(* PLC project Cell Example , CTH FIX1 1.0, author CTH SS2 *)
(* stored: creationDateTime 2009-04-27T15:46:22, companyURL www.chalmers.se, language en-US, organization SS2, modificationDateTime 2008-04-09T20:25:24, version 1.0 *)

PROGRAM EOP10_a
  VAR_EXTERNAL
    Op_10_start : BOOL := false;
    C1C2C1_in_position_empty : BOOL := false;
    C1C2C2_in_off : BOOL := false;
    Op_10_end : BOOL := false;
  END_VAR
  VAR  (* added by the conversion: wires and edge detectors of the diagram *)
    _AND4_OUT : BOOL;
    _AND9_OUT : BOOL;
  END_VAR

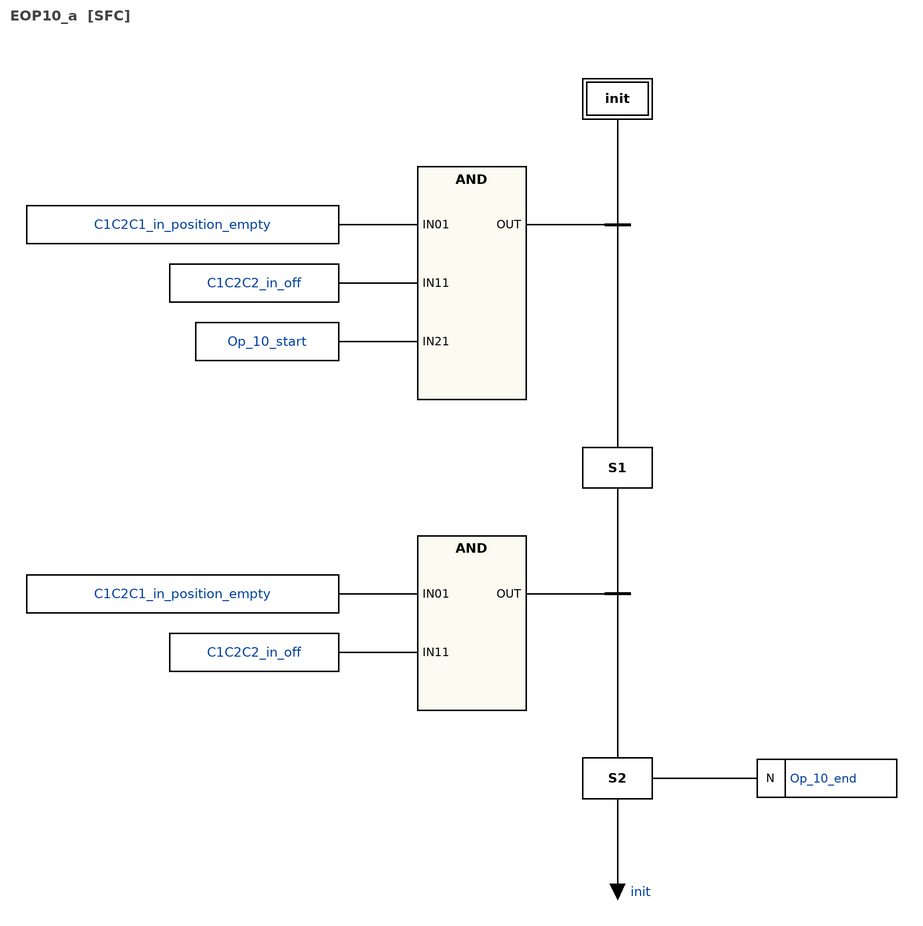
INITIAL_STEP init:
  COMPUTE_FUNCTION_BLOCKS(S);
END_STEP
TRANSITION FROM init TO S1
  := _AND4_OUT;
END_TRANSITION
STEP S1:
END_STEP
TRANSITION FROM S1 TO S2
  := _AND9_OUT;
END_TRANSITION
STEP S2:
  Op_10_end(N);
END_STEP
ACTION COMPUTE_FUNCTION_BLOCKS:  (* blocks drawn on the SFC sheet *)
  _AND4_OUT := C1C2C1_in_position_empty AND C1C2C2_in_off AND Op_10_start;
  _AND9_OUT := C1C2C1_in_position_empty AND C1C2C2_in_off;
END_ACTION
END_PROGRAM

PROGRAM EOP10_b
  VAR_EXTERNAL
    Op_10_start : BOOL := false;
    C1C2C1_in_part_in_position : BOOL := false;
    C1C2C2_in_on : BOOL := false;
    Op_10_end : BOOL := false;
  END_VAR
  VAR  (* added by the conversion: wires and edge detectors of the diagram *)
    _AND4_OUT : BOOL;
    _AND9_OUT : BOOL;
  END_VAR

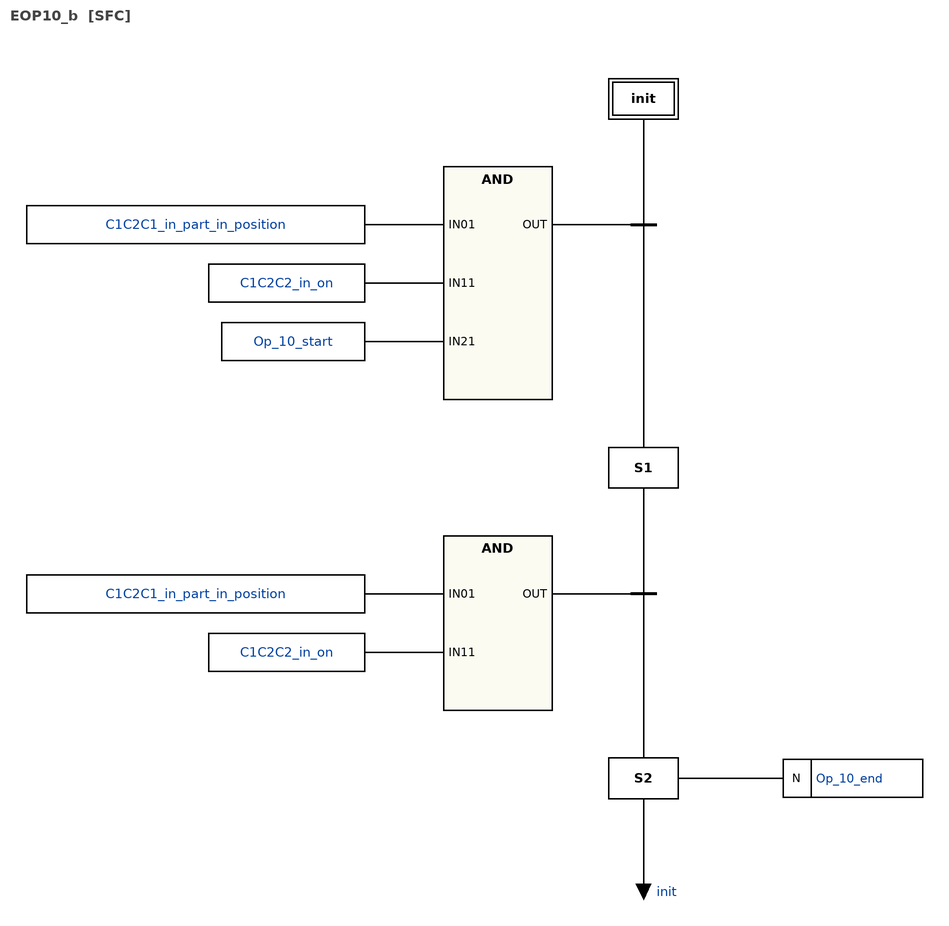
INITIAL_STEP init:
  COMPUTE_FUNCTION_BLOCKS(S);
END_STEP
TRANSITION FROM init TO S1
  := _AND4_OUT;
END_TRANSITION
STEP S1:
END_STEP
TRANSITION FROM S1 TO S2
  := _AND9_OUT;
END_TRANSITION
STEP S2:
  Op_10_end(N);
END_STEP
ACTION COMPUTE_FUNCTION_BLOCKS:  (* blocks drawn on the SFC sheet *)
  _AND4_OUT := C1C2C1_in_part_in_position AND C1C2C2_in_on AND Op_10_start;
  _AND9_OUT := C1C2C1_in_part_in_position AND C1C2C2_in_on;
END_ACTION
END_PROGRAM

PROGRAM EOP11
  VAR_EXTERNAL
    Op_11_start : BOOL := false;
    TRUE_VAR : BOOL := true;
    C1C2_book_zone_1 : BOOL := false;
    C1C2_zone_1_booked : BOOL := false;
    C1C2C1_goto_part_in_position : BOOL := false;
    C1C2C2_goto_on : BOOL := false;
    C1C2C1_in_part_in_position : BOOL := false;
    C1C2C2_in_on : BOOL := false;
    C1C2_unbook_zone_1 : BOOL := false;
    Op_11_end : BOOL := false;
  END_VAR
  VAR  (* added by the conversion: wires and edge detectors of the diagram *)
    _AND14_OUT : BOOL;
    _AND21_OUT : BOOL;
  END_VAR

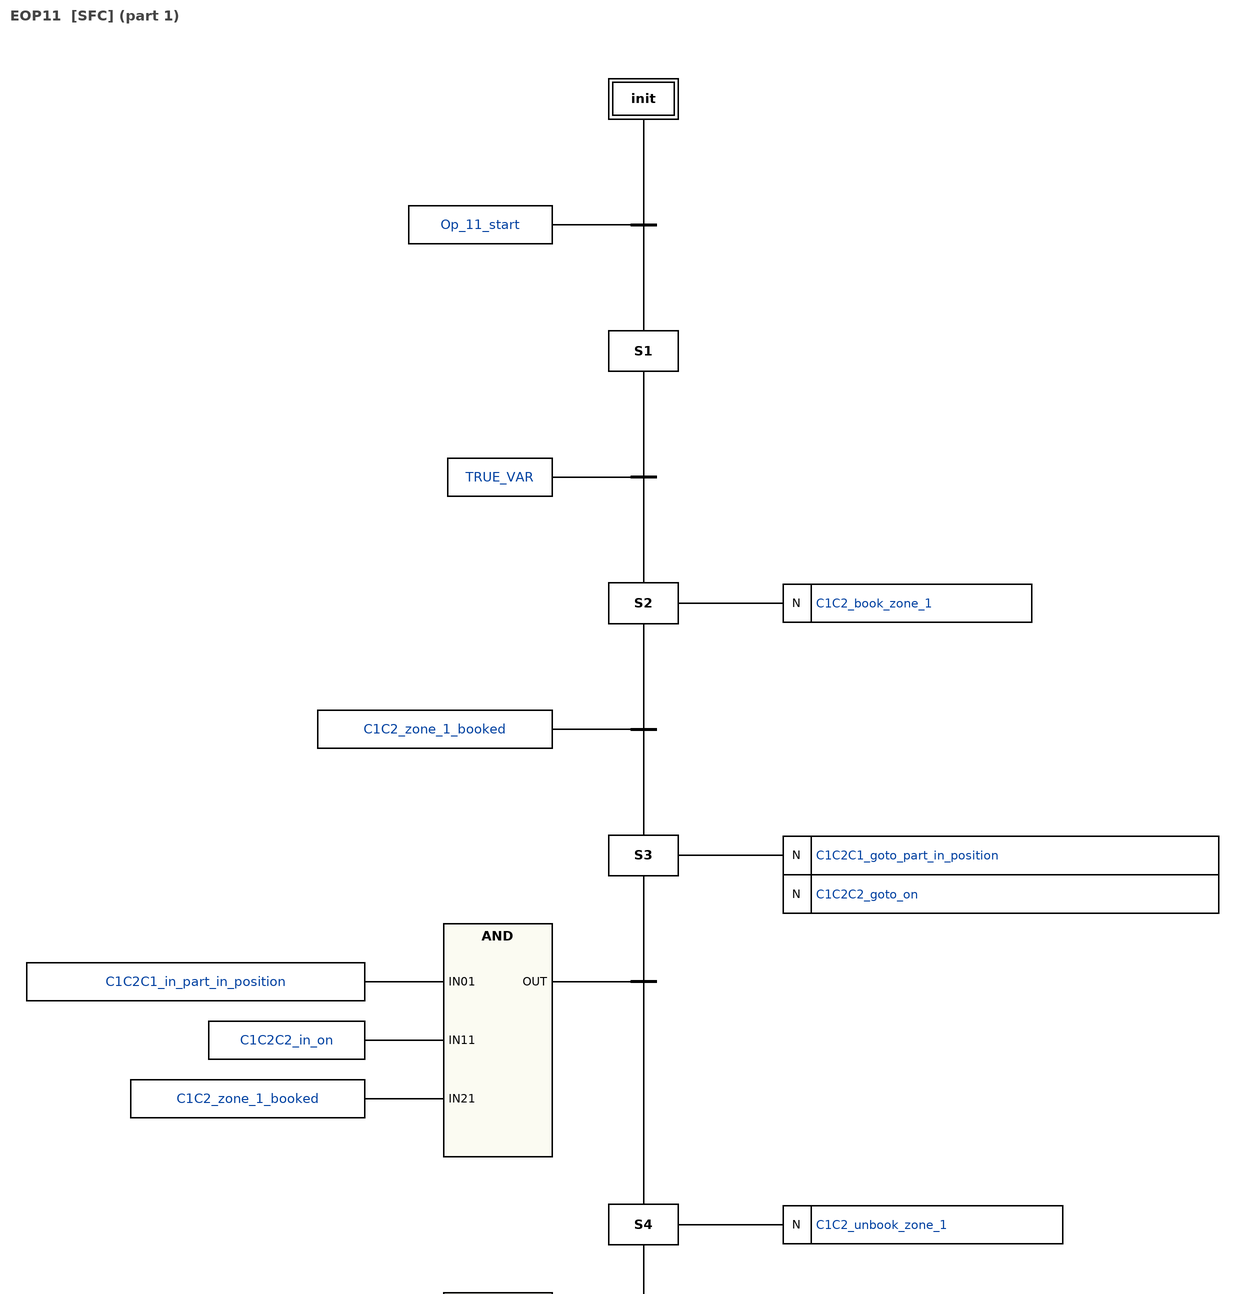
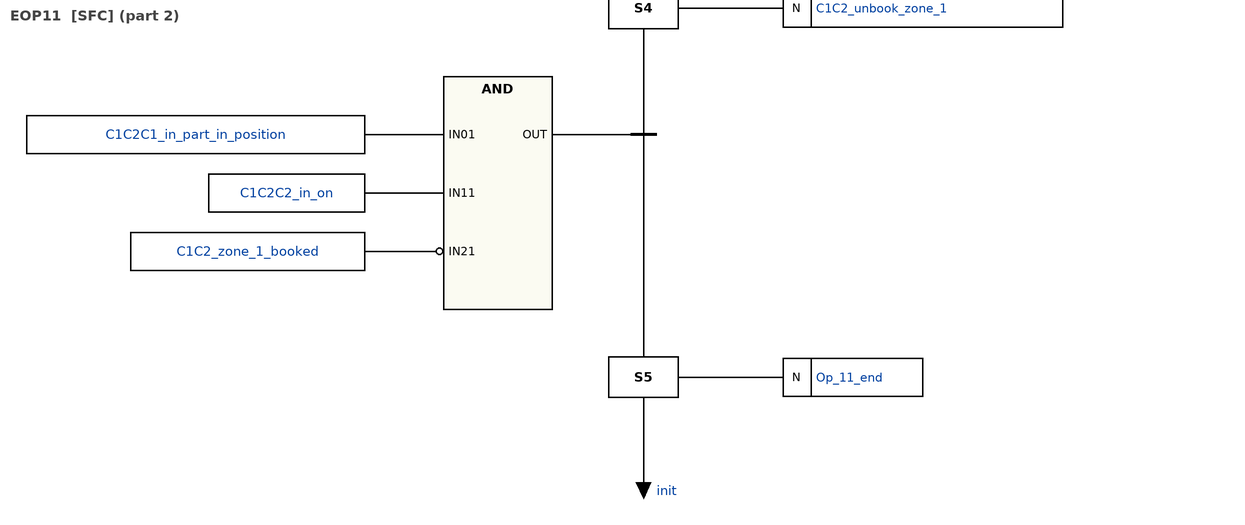
INITIAL_STEP init:
  COMPUTE_FUNCTION_BLOCKS(S);
END_STEP
TRANSITION FROM init TO S1
  := Op_11_start;
END_TRANSITION
STEP S1:
END_STEP
TRANSITION FROM S1 TO S2
  := TRUE_VAR;
END_TRANSITION
STEP S2:
  C1C2_book_zone_1(N);
END_STEP
TRANSITION FROM S2 TO S3
  := C1C2_zone_1_booked;
END_TRANSITION
STEP S3:
  C1C2C1_goto_part_in_position(N);
  C1C2C2_goto_on(N);
END_STEP
TRANSITION FROM S3 TO S4
  := _AND14_OUT;
END_TRANSITION
STEP S4:
  C1C2_unbook_zone_1(N);
END_STEP
TRANSITION FROM S4 TO S5
  := _AND21_OUT;
END_TRANSITION
STEP S5:
  Op_11_end(N);
END_STEP
ACTION COMPUTE_FUNCTION_BLOCKS:  (* blocks drawn on the SFC sheet *)
  _AND14_OUT := C1C2C1_in_part_in_position AND C1C2C2_in_on AND C1C2_zone_1_booked;
  _AND21_OUT := C1C2C1_in_part_in_position AND C1C2C2_in_on AND NOT C1C2_zone_1_booked;
END_ACTION
END_PROGRAM

PROGRAM EOP12
  VAR_EXTERNAL
    Op_12_start : BOOL := false;
    TRUE_VAR : BOOL := true;
    C1C2C1_goto_position_empty : BOOL := false;
    C1C2C2_goto_off : BOOL := false;
    C1C2C1_in_position_empty : BOOL := false;
    C1C2C2_in_off : BOOL := false;
    Op_12_end : BOOL := false;
  END_VAR
  VAR  (* added by the conversion: wires and edge detectors of the diagram *)
    _AND10_OUT : BOOL;
  END_VAR

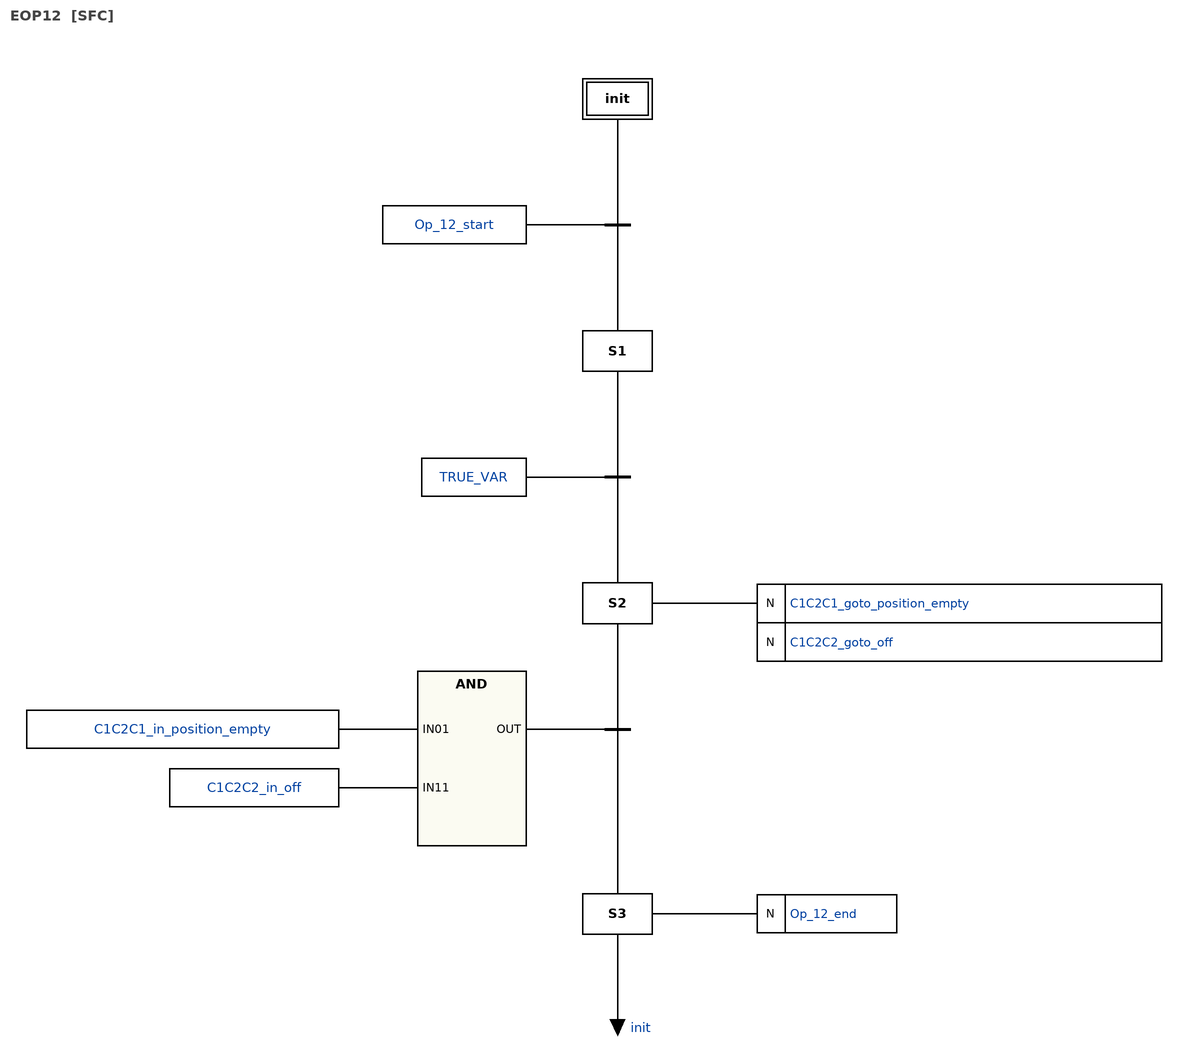
INITIAL_STEP init:
  COMPUTE_FUNCTION_BLOCKS(S);
END_STEP
TRANSITION FROM init TO S1
  := Op_12_start;
END_TRANSITION
STEP S1:
END_STEP
TRANSITION FROM S1 TO S2
  := TRUE_VAR;
END_TRANSITION
STEP S2:
  C1C2C1_goto_position_empty(N);
  C1C2C2_goto_off(N);
END_STEP
TRANSITION FROM S2 TO S3
  := _AND10_OUT;
END_TRANSITION
STEP S3:
  Op_12_end(N);
END_STEP
ACTION COMPUTE_FUNCTION_BLOCKS:  (* blocks drawn on the SFC sheet *)
  _AND10_OUT := C1C2C1_in_position_empty AND C1C2C2_in_off;
END_ACTION
END_PROGRAM

PROGRAM EOP20
  VAR_EXTERNAL
    C1R1_Op20_exe_start : BOOL := false;
    C1R1_in_inital : BOOL := false;
    C1R1_Op20_exe : BOOL := false;
    C1R1_Op20_done : BOOL := false;
  END_VAR

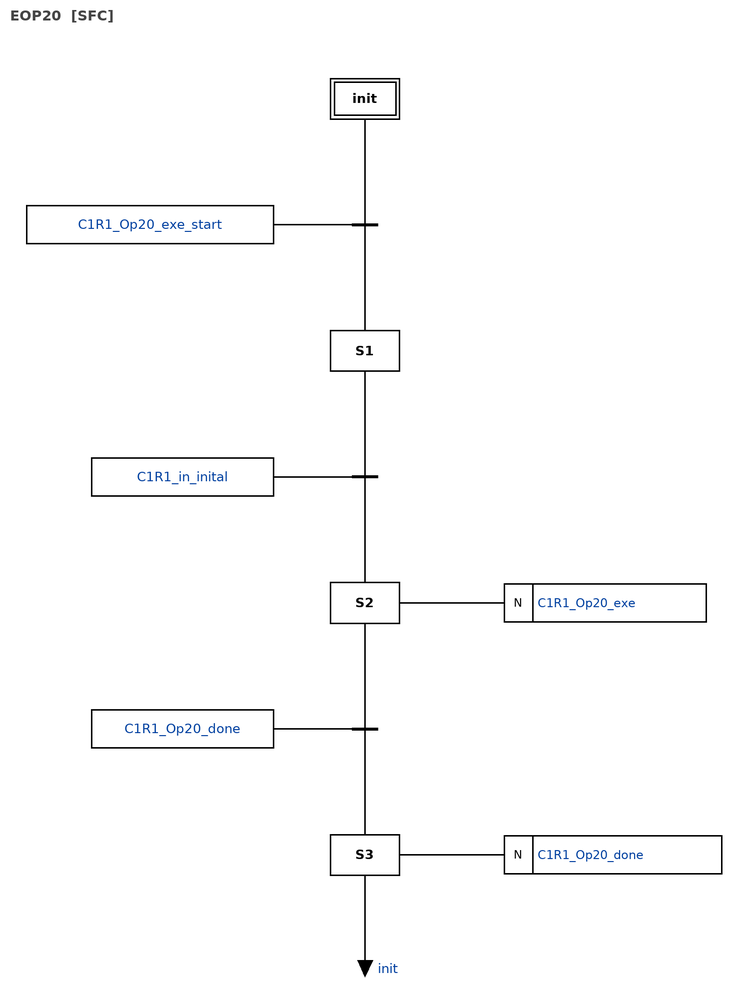
INITIAL_STEP init:
END_STEP
TRANSITION FROM init TO S1
  := C1R1_Op20_exe_start;
END_TRANSITION
STEP S1:
END_STEP
TRANSITION FROM S1 TO S2
  := C1R1_in_inital;
END_TRANSITION
STEP S2:
  C1R1_Op20_exe(N);
END_STEP
TRANSITION FROM S2 TO S3
  := C1R1_Op20_done;
END_TRANSITION
STEP S3:
  C1R1_Op20_done(N);
END_STEP
END_PROGRAM

PROGRAM EOP21
  VAR_EXTERNAL
    C1R1_Op21_exe_start : BOOL := false;
    TRUE_VAR : BOOL := true;
    C1R1_book_zone_1 : BOOL := false;
    C1R1_zone_1_booked : BOOL := false;
    C1R1_Op21_exe : BOOL := false;
    C1R1_Op21_done : BOOL := false;
    C1R1_unbook_zone_1 : BOOL := false;
  END_VAR
  VAR  (* added by the conversion: wires and edge detectors of the diagram *)
    _NOT19_OUT : BOOL;
  END_VAR

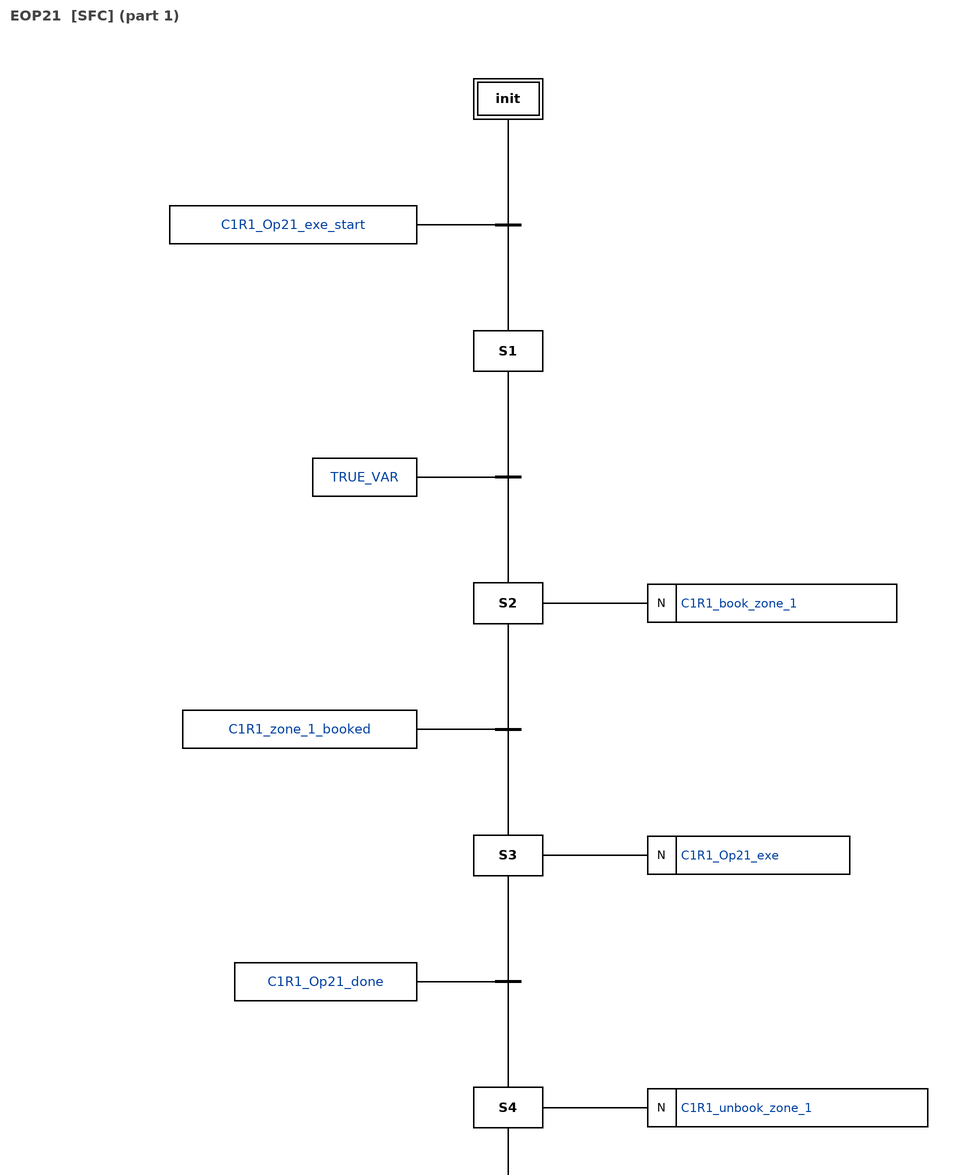
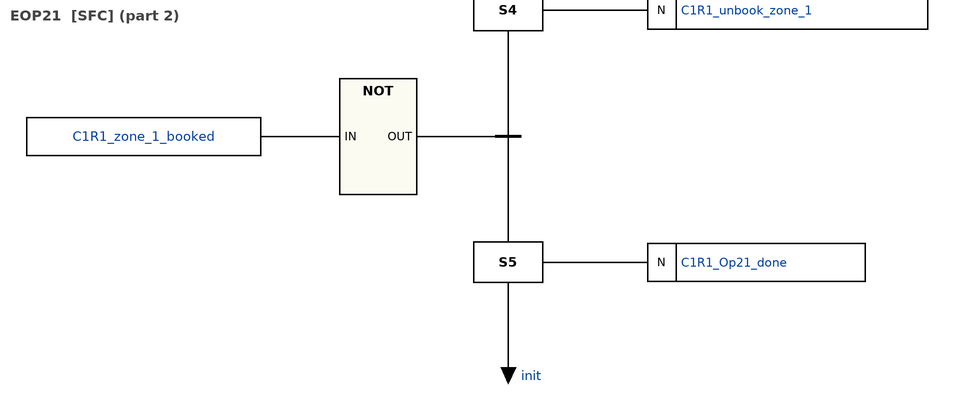
INITIAL_STEP init:
  COMPUTE_FUNCTION_BLOCKS(S);
END_STEP
TRANSITION FROM init TO S1
  := C1R1_Op21_exe_start;
END_TRANSITION
STEP S1:
END_STEP
TRANSITION FROM S1 TO S2
  := TRUE_VAR;
END_TRANSITION
STEP S2:
  C1R1_book_zone_1(N);
END_STEP
TRANSITION FROM S2 TO S3
  := C1R1_zone_1_booked;
END_TRANSITION
STEP S3:
  C1R1_Op21_exe(N);
END_STEP
TRANSITION FROM S3 TO S4
  := C1R1_Op21_done;
END_TRANSITION
STEP S4:
  C1R1_unbook_zone_1(N);
END_STEP
TRANSITION FROM S4 TO S5
  := _NOT19_OUT;
END_TRANSITION
STEP S5:
  C1R1_Op21_done(N);
END_STEP
ACTION COMPUTE_FUNCTION_BLOCKS:  (* blocks drawn on the SFC sheet *)
  _NOT19_OUT := NOT C1R1_zone_1_booked;
END_ACTION
END_PROGRAM

PROGRAM EOP22
  VAR_EXTERNAL
    C1R1_Op22_exe_start : BOOL := false;
    TRUE_VAR : BOOL := true;
    C1R1_book_zone_1 : BOOL := false;
    C1R1_zone_1_booked : BOOL := false;
    C1R1_Op22_exe : BOOL := false;
    C1R1_Op22_done : BOOL := false;
  END_VAR

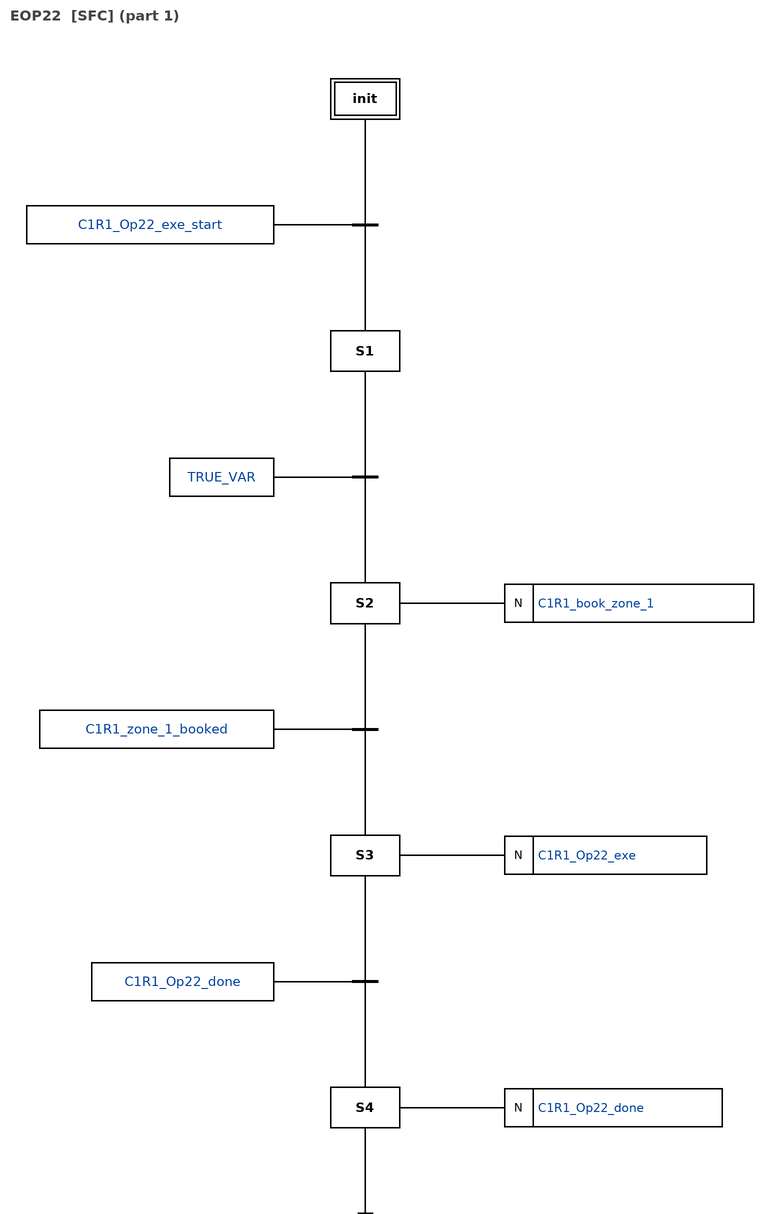
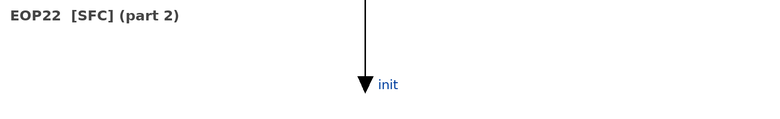
INITIAL_STEP init:
END_STEP
TRANSITION FROM init TO S1
  := C1R1_Op22_exe_start;
END_TRANSITION
STEP S1:
END_STEP
TRANSITION FROM S1 TO S2
  := TRUE_VAR;
END_TRANSITION
STEP S2:
  C1R1_book_zone_1(N);
END_STEP
TRANSITION FROM S2 TO S3
  := C1R1_zone_1_booked;
END_TRANSITION
STEP S3:
  C1R1_Op22_exe(N);
END_STEP
TRANSITION FROM S3 TO S4
  := C1R1_Op22_done;
END_TRANSITION
STEP S4:
  C1R1_Op22_done(N);
END_STEP
END_PROGRAM

PROGRAM EOP23
  VAR_EXTERNAL
    C1R1_Op23_exe_start : BOOL := false;
    TRUE_VAR : BOOL := true;
    C1R1_book_zone_2 : BOOL := false;
    C1R1_zone_2_booked : BOOL := false;
    C1R1_Op23_exe : BOOL := false;
    C1R1_Op23_done : BOOL := false;
    C1R1_unbook_zone_2 : BOOL := false;
  END_VAR
  VAR  (* added by the conversion: wires and edge detectors of the diagram *)
    _NOT19_OUT : BOOL;
  END_VAR

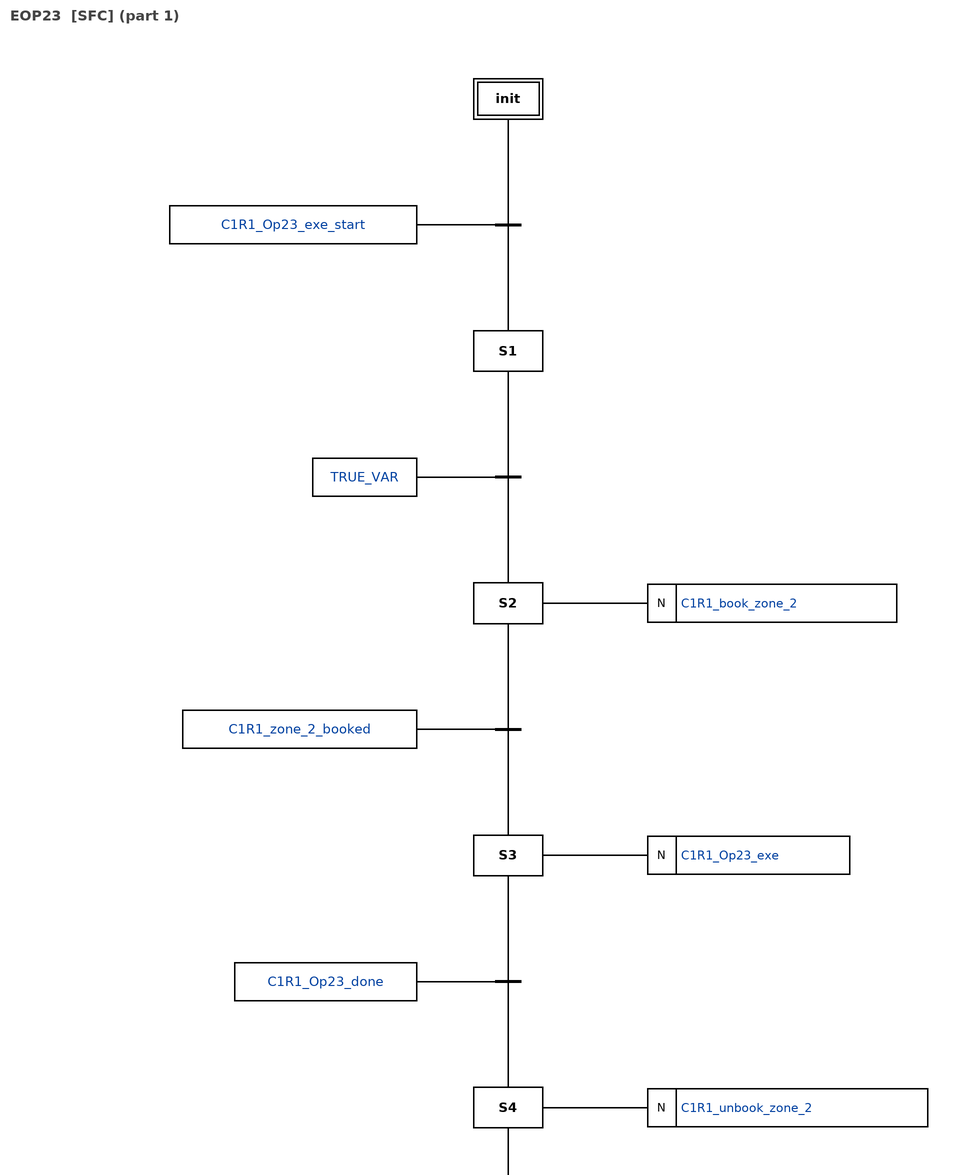
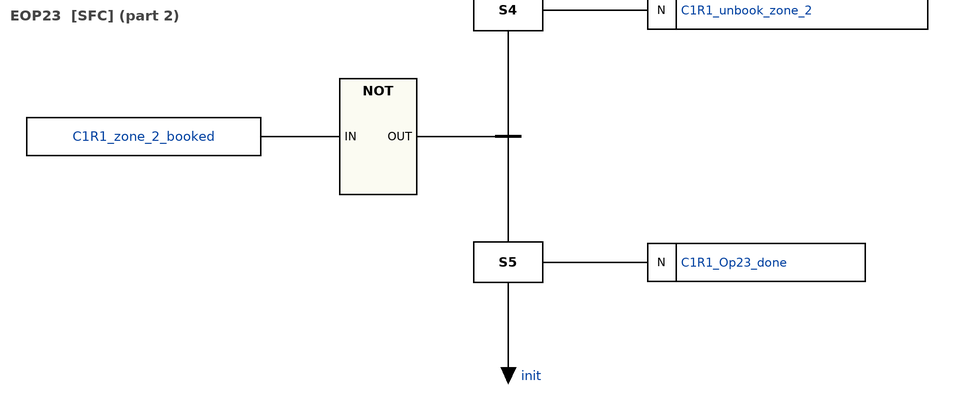
INITIAL_STEP init:
  COMPUTE_FUNCTION_BLOCKS(S);
END_STEP
TRANSITION FROM init TO S1
  := C1R1_Op23_exe_start;
END_TRANSITION
STEP S1:
END_STEP
TRANSITION FROM S1 TO S2
  := TRUE_VAR;
END_TRANSITION
STEP S2:
  C1R1_book_zone_2(N);
END_STEP
TRANSITION FROM S2 TO S3
  := C1R1_zone_2_booked;
END_TRANSITION
STEP S3:
  C1R1_Op23_exe(N);
END_STEP
TRANSITION FROM S3 TO S4
  := C1R1_Op23_done;
END_TRANSITION
STEP S4:
  C1R1_unbook_zone_2(N);
END_STEP
TRANSITION FROM S4 TO S5
  := _NOT19_OUT;
END_TRANSITION
STEP S5:
  C1R1_Op23_done(N);
END_STEP
ACTION COMPUTE_FUNCTION_BLOCKS:  (* blocks drawn on the SFC sheet *)
  _NOT19_OUT := NOT C1R1_zone_2_booked;
END_ACTION
END_PROGRAM

PROGRAM EOP24
  VAR_EXTERNAL
    C1R1_Op24_exe_start : BOOL := false;
    TRUE_VAR : BOOL := true;
    C1R1_book_zone_3 : BOOL := false;
    C1R1_zone_3_booked : BOOL := false;
    C1R1_Op24_exe : BOOL := false;
    C1R1_Op24_done : BOOL := false;
    C1R1_unbook_zone_3 : BOOL := false;
  END_VAR
  VAR  (* added by the conversion: wires and edge detectors of the diagram *)
    _NOT19_OUT : BOOL;
  END_VAR

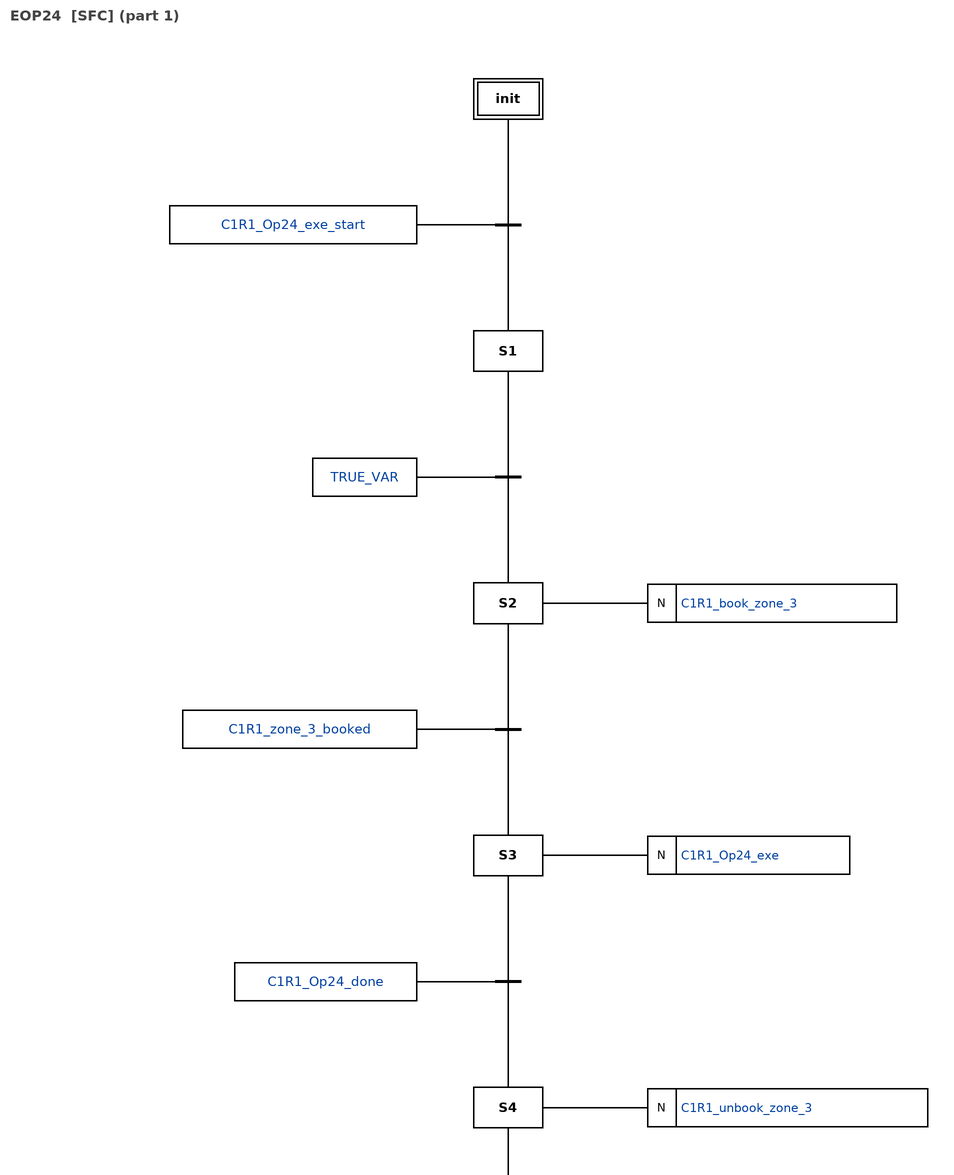
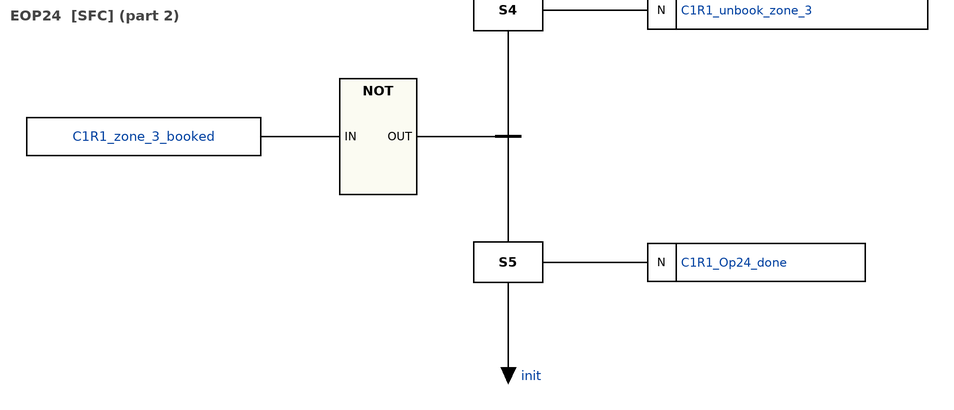
INITIAL_STEP init:
  COMPUTE_FUNCTION_BLOCKS(S);
END_STEP
TRANSITION FROM init TO S1
  := C1R1_Op24_exe_start;
END_TRANSITION
STEP S1:
END_STEP
TRANSITION FROM S1 TO S2
  := TRUE_VAR;
END_TRANSITION
STEP S2:
  C1R1_book_zone_3(N);
END_STEP
TRANSITION FROM S2 TO S3
  := C1R1_zone_3_booked;
END_TRANSITION
STEP S3:
  C1R1_Op24_exe(N);
END_STEP
TRANSITION FROM S3 TO S4
  := C1R1_Op24_done;
END_TRANSITION
STEP S4:
  C1R1_unbook_zone_3(N);
END_STEP
TRANSITION FROM S4 TO S5
  := _NOT19_OUT;
END_TRANSITION
STEP S5:
  C1R1_Op24_done(N);
END_STEP
ACTION COMPUTE_FUNCTION_BLOCKS:  (* blocks drawn on the SFC sheet *)
  _NOT19_OUT := NOT C1R1_zone_3_booked;
END_ACTION
END_PROGRAM

PROGRAM EOP30
  VAR_EXTERNAL
    Op_30_start : BOOL := false;
    C1F1C1_in_home : BOOL := false;
    C1F1C2_in_locked : BOOL := false;
    C1F1C3_in_open : BOOL := false;
    C1F1C4_in_off : BOOL := false;
    Op_30_end : BOOL := false;
  END_VAR
  VAR  (* added by the conversion: wires and edge detectors of the diagram *)
    _AND6_OUT : BOOL;
  END_VAR

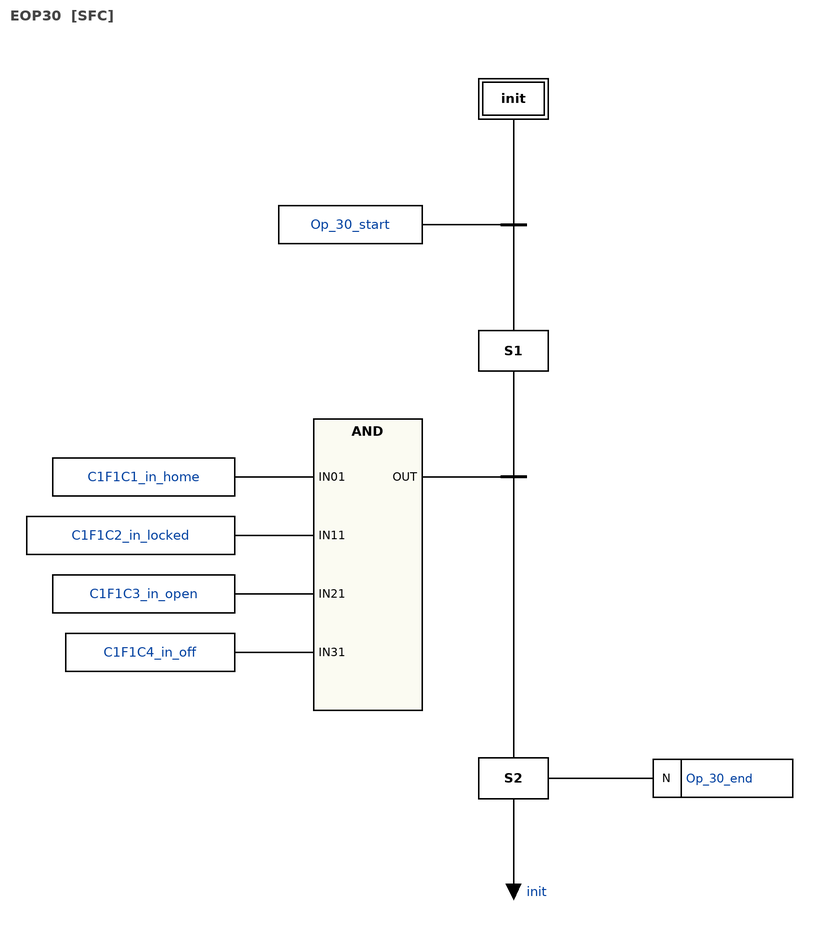
INITIAL_STEP init:
  COMPUTE_FUNCTION_BLOCKS(S);
END_STEP
TRANSITION FROM init TO S1
  := Op_30_start;
END_TRANSITION
STEP S1:
END_STEP
TRANSITION FROM S1 TO S2
  := _AND6_OUT;
END_TRANSITION
STEP S2:
  Op_30_end(N);
END_STEP
ACTION COMPUTE_FUNCTION_BLOCKS:  (* blocks drawn on the SFC sheet *)
  _AND6_OUT := C1F1C1_in_home AND C1F1C2_in_locked AND C1F1C3_in_open AND C1F1C4_in_off;
END_ACTION
END_PROGRAM

PROGRAM EOP31
  VAR_EXTERNAL
    Op_31_start : BOOL := false;
    TRUE_VAR : BOOL := true;
    Op_31_end : BOOL := false;
  END_VAR

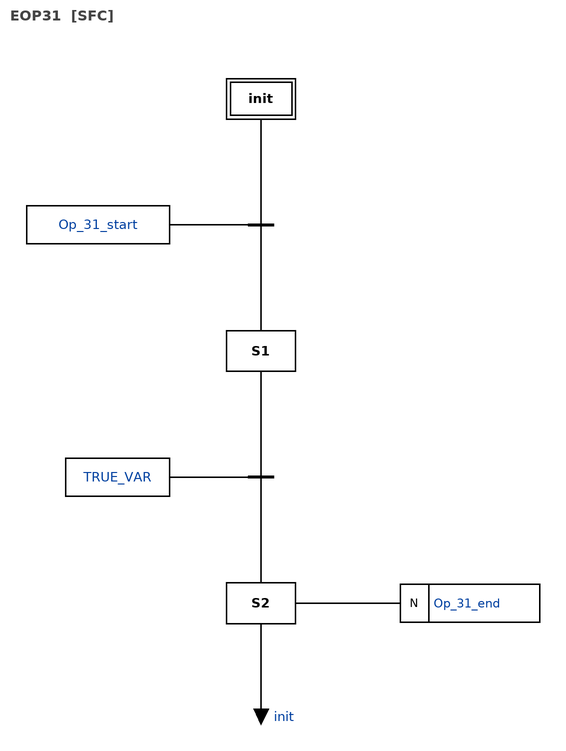
INITIAL_STEP init:
END_STEP
TRANSITION FROM init TO S1
  := Op_31_start;
END_TRANSITION
STEP S1:
END_STEP
TRANSITION FROM S1 TO S2
  := TRUE_VAR;
END_TRANSITION
STEP S2:
  Op_31_end(N);
END_STEP
END_PROGRAM

PROGRAM EOP32
  VAR_EXTERNAL
    Op_32_start : BOOL := false;
    TRUE_VAR : BOOL := true;
    C1F1C1_goto_home : BOOL := false;
    C1F1C2_goto_locked : BOOL := false;
    C1F1C3_goto_close : BOOL := false;
    C1F1C4_goto_on : BOOL := false;
    C1F1C1_in_home : BOOL := false;
    C1F1C2_in_locked : BOOL := false;
    C1F1C3_in_close : BOOL := false;
    C1F1C4_in_on : BOOL := false;
    Op_32_end : BOOL := false;
  END_VAR
  VAR  (* added by the conversion: wires and edge detectors of the diagram *)
    _AND10_OUT : BOOL;
  END_VAR

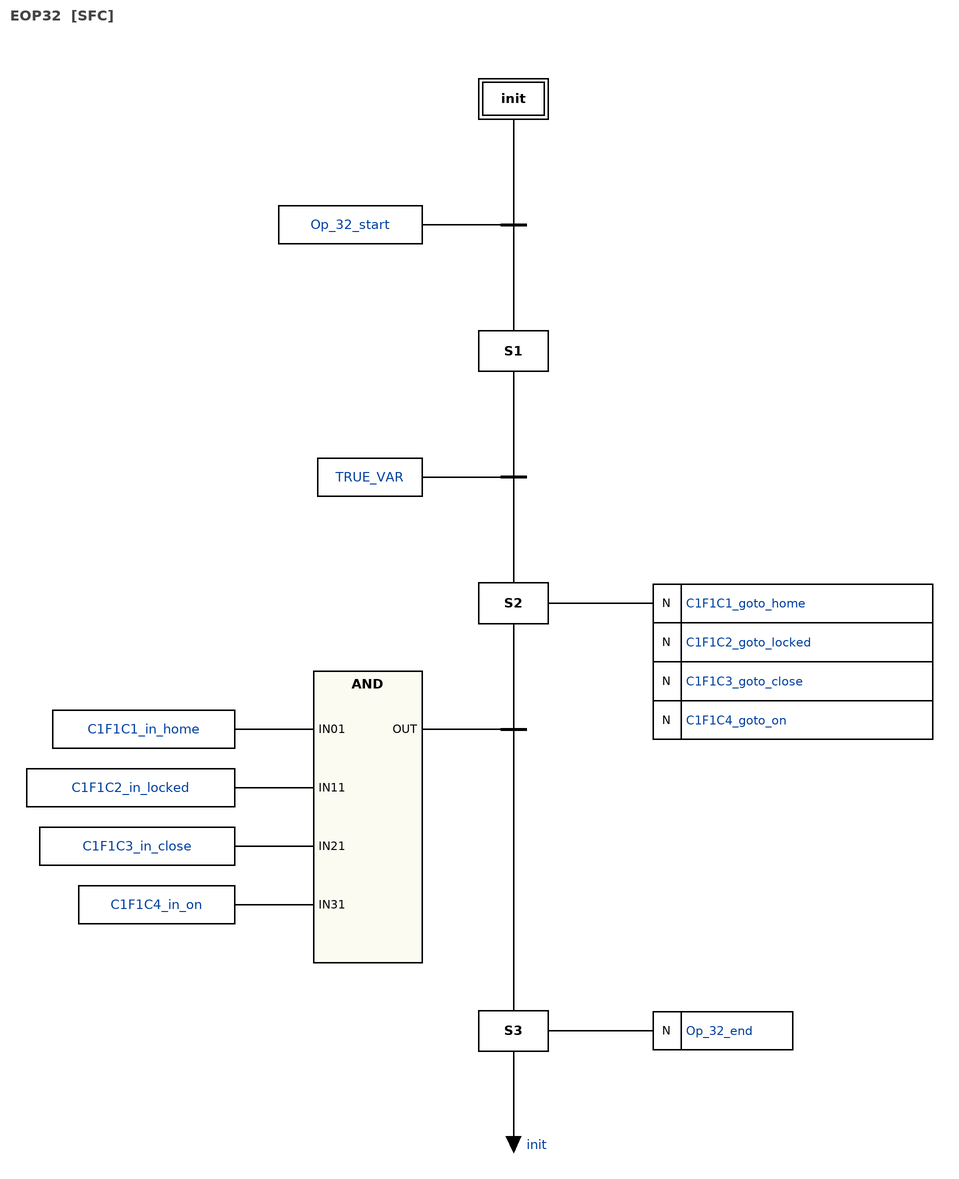
INITIAL_STEP init:
  COMPUTE_FUNCTION_BLOCKS(S);
END_STEP
TRANSITION FROM init TO S1
  := Op_32_start;
END_TRANSITION
STEP S1:
END_STEP
TRANSITION FROM S1 TO S2
  := TRUE_VAR;
END_TRANSITION
STEP S2:
  C1F1C1_goto_home(N);
  C1F1C2_goto_locked(N);
  C1F1C3_goto_close(N);
  C1F1C4_goto_on(N);
END_STEP
TRANSITION FROM S2 TO S3
  := _AND10_OUT;
END_TRANSITION
STEP S3:
  Op_32_end(N);
END_STEP
ACTION COMPUTE_FUNCTION_BLOCKS:  (* blocks drawn on the SFC sheet *)
  _AND10_OUT := C1F1C1_in_home AND C1F1C2_in_locked AND C1F1C3_in_close AND C1F1C4_in_on;
END_ACTION
END_PROGRAM

PROGRAM EOP33
  VAR_EXTERNAL
    Op_33_start : BOOL := false;
    TRUE_VAR : BOOL := true;
    C1F1C1_goto_home : BOOL := false;
    C1F1C2_goto_unlocked : BOOL := false;
    C1F1C3_goto_close : BOOL := false;
    C1F1C4_goto_on : BOOL := false;
    C1F1_book_zone_2 : BOOL := false;
    C1F1_book_zone_3 : BOOL := false;
    C1F1C1_in_home : BOOL := false;
    C1F1C2_in_unlocked : BOOL := false;
    C1F1C3_in_close : BOOL := false;
    C1F1C4_in_on : BOOL := false;
    C1F1_zone_2_booked : BOOL := false;
    C1F1_zone_3_booked : BOOL := false;
    C1F1C1_goto_work_pos : BOOL := false;
    C1F1C1_in_work_pos : BOOL := false;
    C1F1C2_goto_locked : BOOL := false;
    C1F1_unbook_zone_3 : BOOL := false;
    C1F1C2_in_locked : BOOL := false;
    Op_33_end : BOOL := false;
  END_VAR
  VAR  (* added by the conversion: wires and edge detectors of the diagram *)
    _AND10_OUT : BOOL;
    _AND20_OUT : BOOL;
    _AND30_OUT : BOOL;
  END_VAR

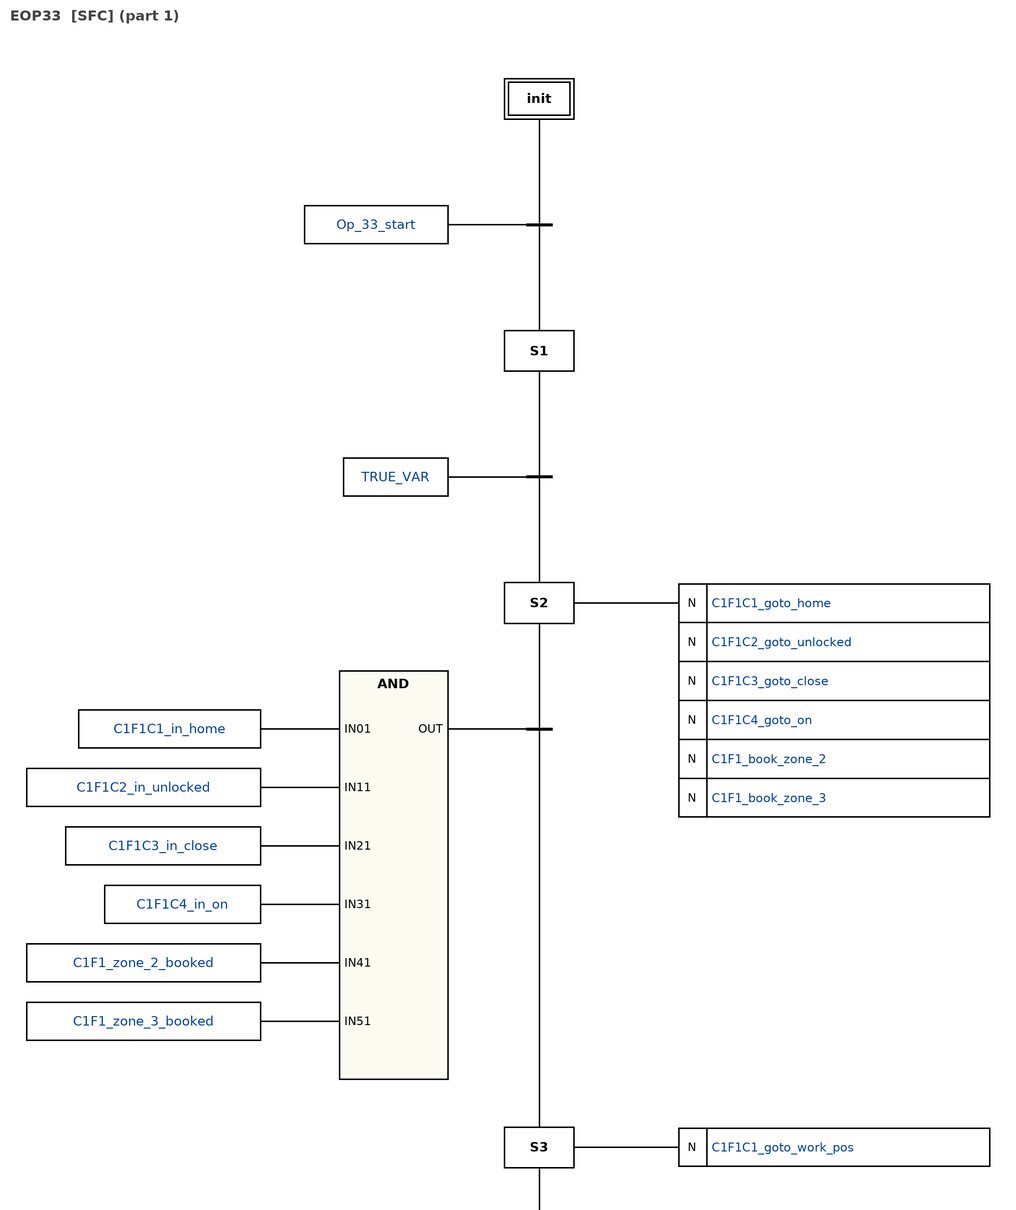
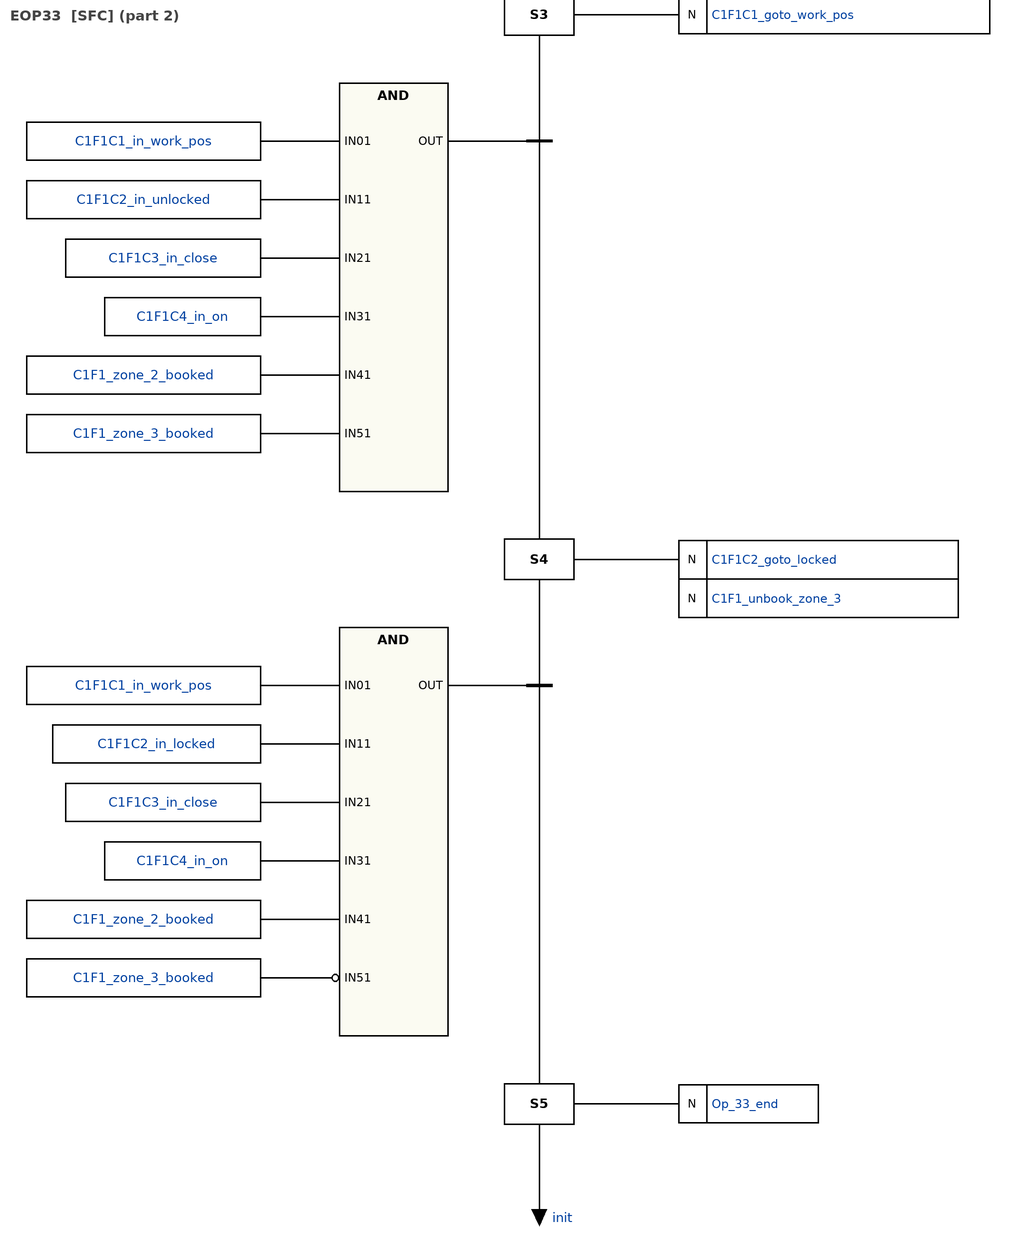
INITIAL_STEP init:
  COMPUTE_FUNCTION_BLOCKS(S);
END_STEP
TRANSITION FROM init TO S1
  := Op_33_start;
END_TRANSITION
STEP S1:
END_STEP
TRANSITION FROM S1 TO S2
  := TRUE_VAR;
END_TRANSITION
STEP S2:
  C1F1C1_goto_home(N);
  C1F1C2_goto_unlocked(N);
  C1F1C3_goto_close(N);
  C1F1C4_goto_on(N);
  C1F1_book_zone_2(N);
  C1F1_book_zone_3(N);
END_STEP
TRANSITION FROM S2 TO S3
  := _AND10_OUT;
END_TRANSITION
STEP S3:
  C1F1C1_goto_work_pos(N);
END_STEP
TRANSITION FROM S3 TO S4
  := _AND20_OUT;
END_TRANSITION
STEP S4:
  C1F1C2_goto_locked(N);
  C1F1_unbook_zone_3(N);
END_STEP
TRANSITION FROM S4 TO S5
  := _AND30_OUT;
END_TRANSITION
STEP S5:
  Op_33_end(N);
END_STEP
ACTION COMPUTE_FUNCTION_BLOCKS:  (* blocks drawn on the SFC sheet *)
  _AND10_OUT := C1F1C1_in_home AND C1F1C2_in_unlocked AND C1F1C3_in_close AND C1F1C4_in_on AND C1F1_zone_2_booked AND C1F1_zone_3_booked;
  _AND20_OUT := C1F1C1_in_work_pos AND C1F1C2_in_unlocked AND C1F1C3_in_close AND C1F1C4_in_on AND C1F1_zone_2_booked AND C1F1_zone_3_booked;
  _AND30_OUT := C1F1C1_in_work_pos AND C1F1C2_in_locked AND C1F1C3_in_close AND C1F1C4_in_on AND C1F1_zone_2_booked AND NOT C1F1_zone_3_booked;
END_ACTION
END_PROGRAM

PROGRAM EOP34
  VAR_EXTERNAL
    Op_34_start : BOOL := false;
    TRUE_VAR : BOOL := true;
    C1F1C1_goto_work_pos : BOOL := false;
    C1F1C2_goto_locked : BOOL := false;
    C1F1C3_goto_open : BOOL := false;
    C1F1C4_goto_on : BOOL := false;
    C1F1_book_zone_2 : BOOL := false;
    C1F1C1_in_work_pos : BOOL := false;
    C1F1C2_in_locked : BOOL := false;
    C1F1C3_in_open : BOOL := false;
    C1F1C4_in_on : BOOL := false;
    C1F1_zone_2_booked : BOOL := false;
    C1F1C2_goto_unlocked : BOOL := false;
    C1F1C2_in_unlocked : BOOL := false;
    C1F1C1_goto_home : BOOL := false;
    C1F1C4_goto_off : BOOL := false;
    C1F1C1_in_home : BOOL := false;
    C1F1C4_in_off : BOOL := false;
    C1F1_unbook_zone_2 : BOOL := false;
    Op_34_end : BOOL := false;
  END_VAR
  VAR  (* added by the conversion: wires and edge detectors of the diagram *)
    _AND10_OUT : BOOL;
    _AND19_OUT : BOOL;
    _AND28_OUT : BOOL;
    _AND37_OUT : BOOL;
  END_VAR

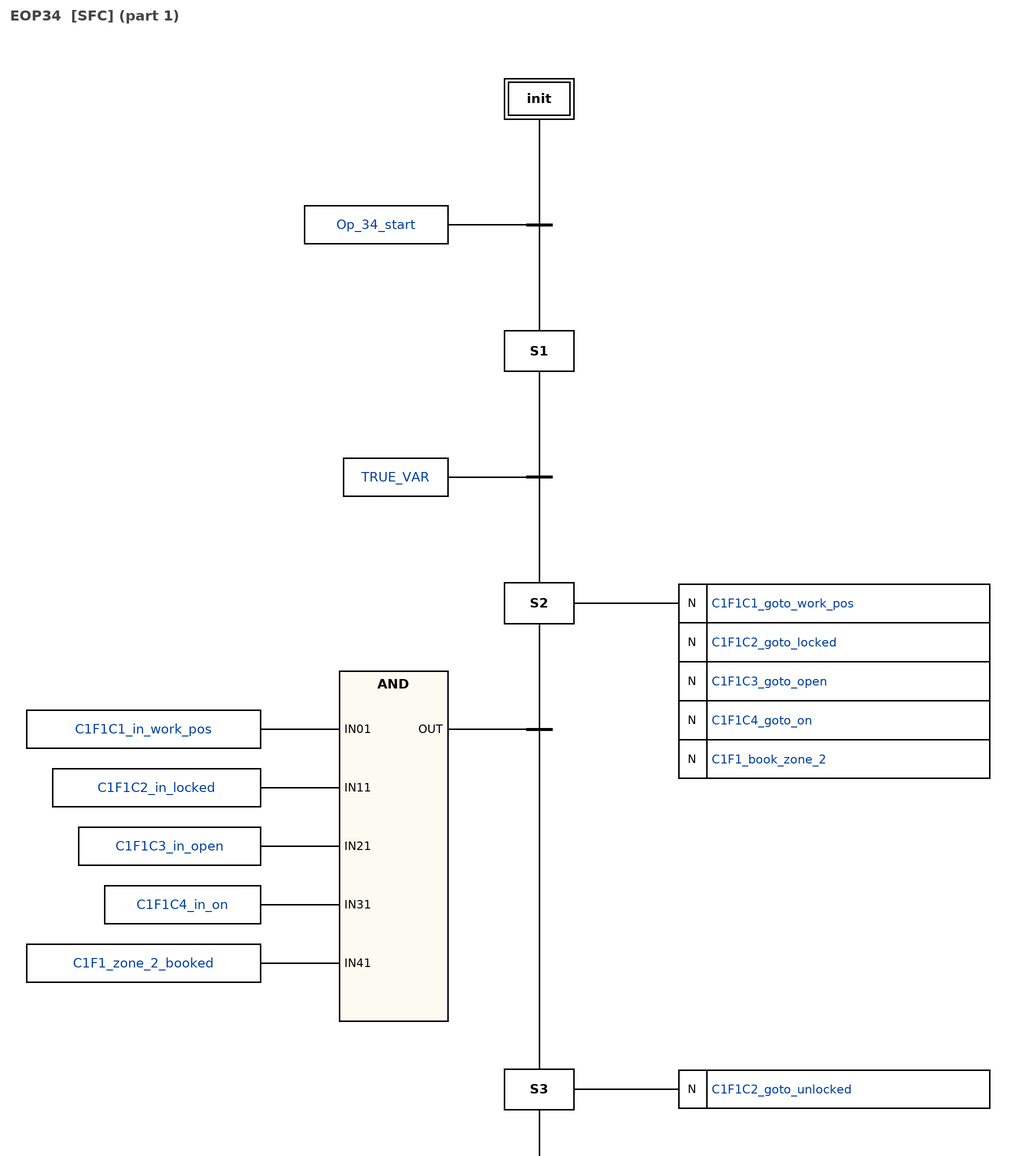
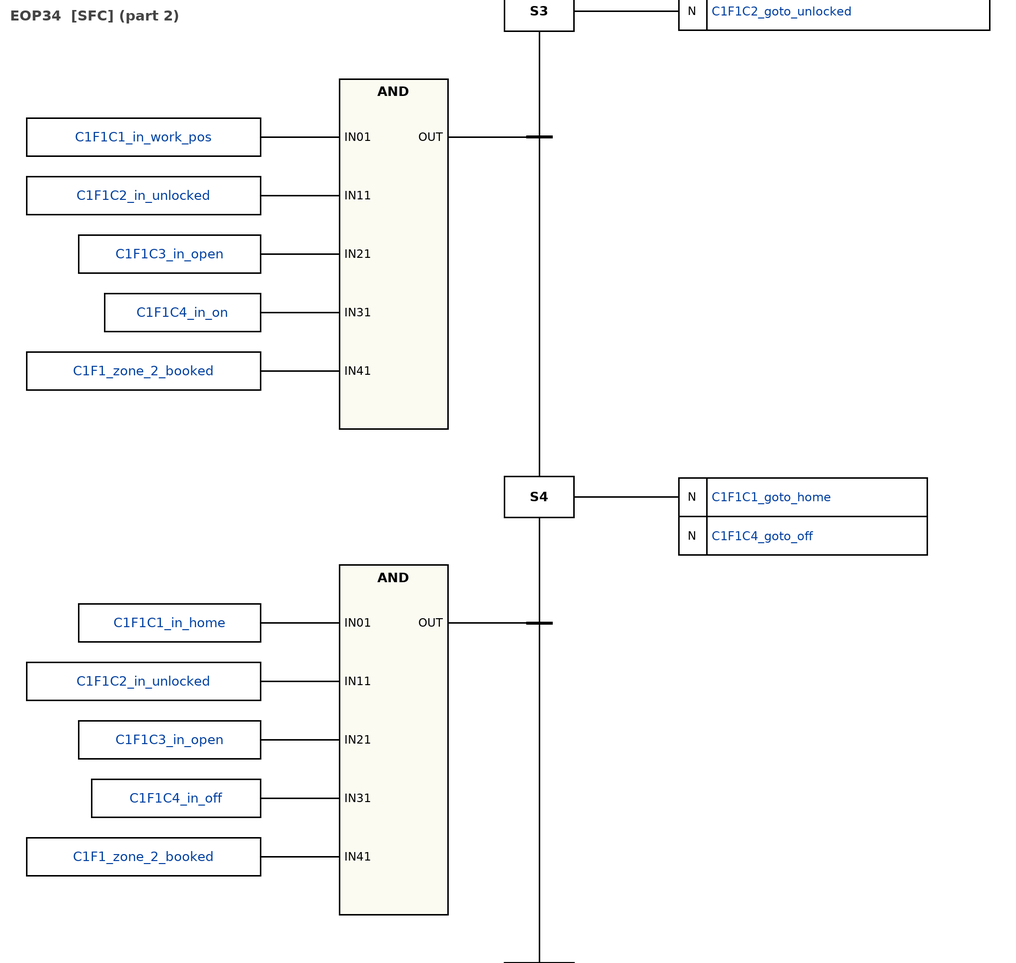
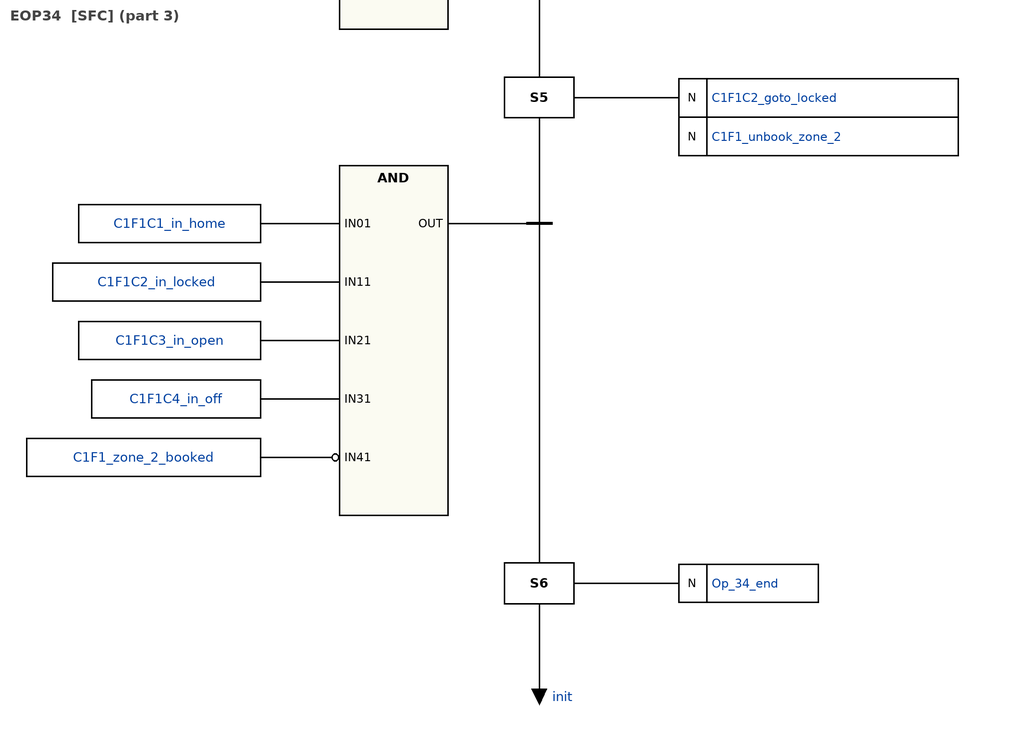
INITIAL_STEP init:
  COMPUTE_FUNCTION_BLOCKS(S);
END_STEP
TRANSITION FROM init TO S1
  := Op_34_start;
END_TRANSITION
STEP S1:
END_STEP
TRANSITION FROM S1 TO S2
  := TRUE_VAR;
END_TRANSITION
STEP S2:
  C1F1C1_goto_work_pos(N);
  C1F1C2_goto_locked(N);
  C1F1C3_goto_open(N);
  C1F1C4_goto_on(N);
  C1F1_book_zone_2(N);
END_STEP
TRANSITION FROM S2 TO S3
  := _AND10_OUT;
END_TRANSITION
STEP S3:
  C1F1C2_goto_unlocked(N);
END_STEP
TRANSITION FROM S3 TO S4
  := _AND19_OUT;
END_TRANSITION
STEP S4:
  C1F1C1_goto_home(N);
  C1F1C4_goto_off(N);
END_STEP
TRANSITION FROM S4 TO S5
  := _AND28_OUT;
END_TRANSITION
STEP S5:
  C1F1C2_goto_locked(N);
  C1F1_unbook_zone_2(N);
END_STEP
TRANSITION FROM S5 TO S6
  := _AND37_OUT;
END_TRANSITION
STEP S6:
  Op_34_end(N);
END_STEP
ACTION COMPUTE_FUNCTION_BLOCKS:  (* blocks drawn on the SFC sheet *)
  _AND10_OUT := C1F1C1_in_work_pos AND C1F1C2_in_locked AND C1F1C3_in_open AND C1F1C4_in_on AND C1F1_zone_2_booked;
  _AND19_OUT := C1F1C1_in_work_pos AND C1F1C2_in_unlocked AND C1F1C3_in_open AND C1F1C4_in_on AND C1F1_zone_2_booked;
  _AND28_OUT := C1F1C1_in_home AND C1F1C2_in_unlocked AND C1F1C3_in_open AND C1F1C4_in_off AND C1F1_zone_2_booked;
  _AND37_OUT := C1F1C1_in_home AND C1F1C2_in_locked AND C1F1C3_in_open AND C1F1C4_in_off AND NOT C1F1_zone_2_booked;
END_ACTION
END_PROGRAM

PROGRAM EOP40
  VAR_EXTERNAL
    C1C1_Op40_exe_start : BOOL := false;
    TRUE_VAR : BOOL := true;
    C1C1_Op40_done : BOOL := false;
  END_VAR

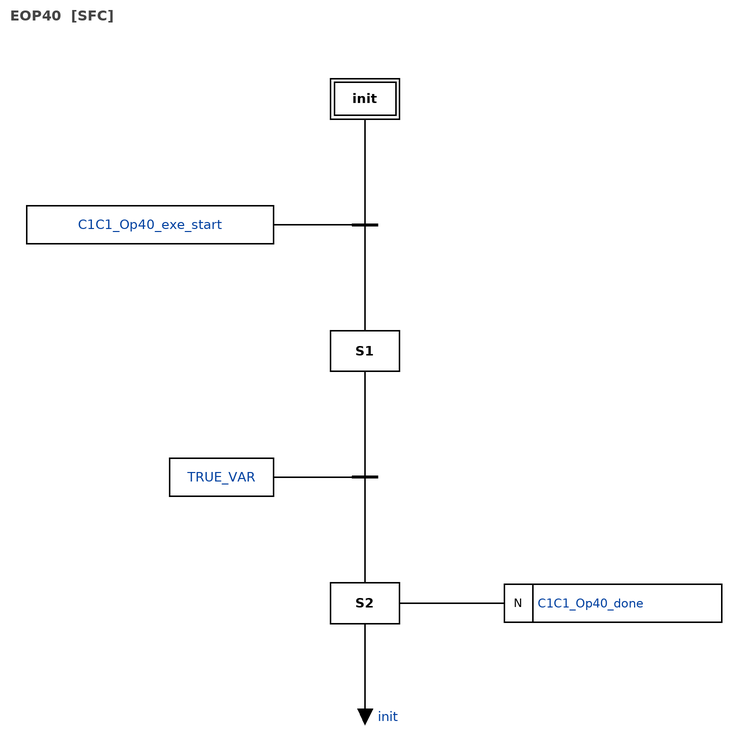
INITIAL_STEP init:
END_STEP
TRANSITION FROM init TO S1
  := C1C1_Op40_exe_start;
END_TRANSITION
STEP S1:
END_STEP
TRANSITION FROM S1 TO S2
  := TRUE_VAR;
END_TRANSITION
STEP S2:
  C1C1_Op40_done(N);
END_STEP
END_PROGRAM

PROGRAM EOP41
  VAR_EXTERNAL
    C1C1_Op41_exe_start : BOOL := false;
    TRUE_VAR : BOOL := true;
    C1C1_book_zone_2 : BOOL := false;
    C1C1_book_zone_3 : BOOL := false;
    C1C1_zone_2_booked : BOOL := false;
    C1C1_zone_3_booked : BOOL := false;
    C1C1C1_goto_unprocessed : BOOL := false;
    C1C1C1_in_unprocessed : BOOL := false;
    C1C1_unbook_zone_2 : BOOL := false;
    C1C1_unbook_zone_3 : BOOL := false;
    C1C1_Op41_done : BOOL := false;
  END_VAR
  VAR  (* added by the conversion: wires and edge detectors of the diagram *)
    _AND10_OUT : BOOL;
    _AND16_OUT : BOOL;
    _AND23_OUT : BOOL;
  END_VAR

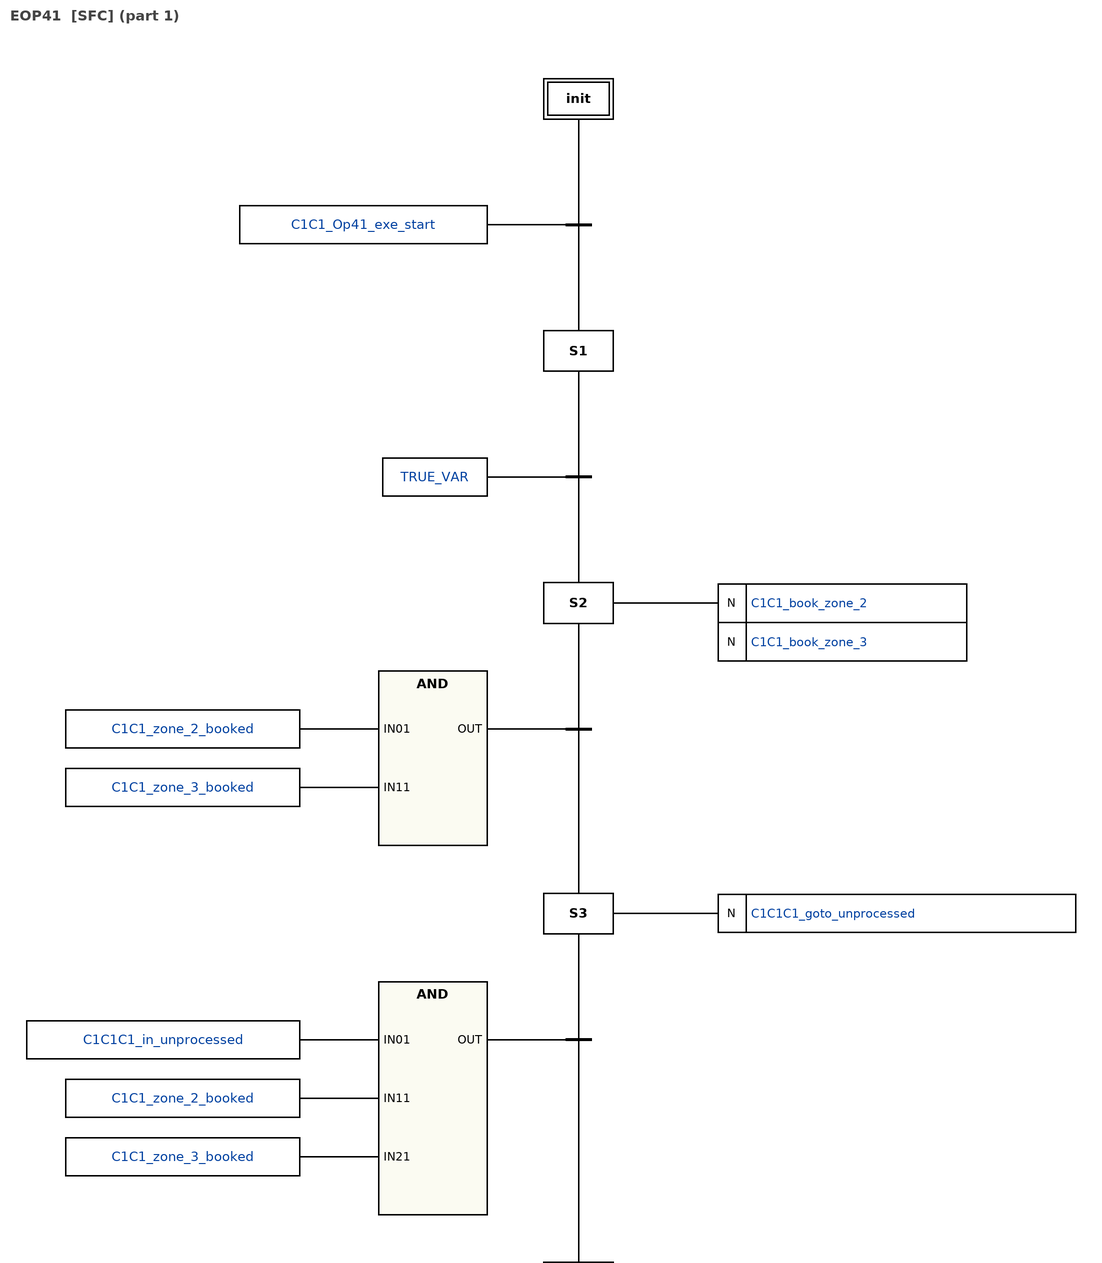
